# EPICS substitutions: motionSetPointsApp/Db/motionSetPointsDoubleAxis.substitutions
file "$(TOP)/motionSetPointsApp/Db/motionSetPointsHeader.template" {
	pattern{ P, LOOKUP, AXIS1, AXIS2 }
	{ "\$(P)", "\$(LOOKUP)", "\$(AXIS1)", "\$(AXIS2)" }
}

file "$(TOP)/motionSetPointsApp/Db/single_axis.template" {
	pattern{ P, AXIS_NUM, AXIS, LOOKUP }
	{ "\$(P)", "0", "\$(AXIS1)", "\$(LOOKUP)" }
	{ "\$(P)", "1", "\$(AXIS2)", "\$(LOOKUP)" }
}
